{attribute 'linkalways'} 
{attribute 'no_explicit_call' := 'This FB is a CLASS and must be accessed using methods or properties'}
{attribute 'enable_dynamic_creation'}
FUNCTION_BLOCK _ALIASTYP EXTENDS AliasDatatypeBase
VAR
	localData : ALIASTYP;
	activeData : REFERENCE TO ALIASTYP REF= localData;
	aliasBaseDatatype : ALIASTYPBASE;
END_VAR

PROPERTY PUBLIC Address : PVOID
GET
Address := ADR(activeData);
END_GET
END_PROPERTY

METHOD PUBLIC ClearReference
VAR_INPUT
END_VAR
activeData REF= localData;
SetBaseDatatypeReference();
END_METHOD

METHOD PUBLIC Clone : I_Datatype
VAR
    pClone : POINTER TO _ALIASTYP;
END_VAR
pClone := __NEW(_ALIASTYP);
Clone := pClone^;
END_METHOD

METHOD FB_init : BOOL
VAR_INPUT
	bInitRetains : BOOL; // if TRUE, the retain variables are initialized (warm start / cold start)
	bInCopyCode : BOOL;  // if TRUE, the instance afterwards gets moved into the copy code (online change)
	//InitialValue : ALIASTYP; // if possible, not all values can be initialized
END_VAR
//localData := InitialValue; // if possible, not all values can be initialized
SetBaseDatatypeReference();
AddBaseDatatype(aliasBaseDatatype);
END_METHOD

PROPERTY PUBLIC Identifier : T_MAXSTRING
GET
Identifier := 'ALIASTYP';
END_GET
END_PROPERTY

METHOD PUBLIC MakeReferenceTo
VAR_INPUT
	ReferenceTarget : REFERENCE TO ALIASTYP;
END_VAR
activeData REF= ReferenceTarget;
SetBaseDatatypeReference();
END_METHOD

METHOD PROTECTED SetBaseDatatypeReference
VAR_INPUT
END_VAR
aliasBaseDatatype.MakeReferenceTo(activeData);
END_METHOD

PROPERTY PUBLIC Size : UDINT
GET
Size := SIZEOF(activeData);
END_GET
END_PROPERTY

METHOD TryMakeReferenceTo : BOOL
VAR_INPUT
	Target : I_Datatype;
END_VAR
VAR
	pTargetData : POINTER TO ALIASTYP;
END_VAR
IF NOT IsEquivalentTo(Target) THEN
	RETURN;
END_IF

pTargetData := Target.Address;
activeData REF= pTargetData^;
SetBaseDatatypeReference();
TryMakeReferenceTo := TRUE;
END_METHOD

PROPERTY PUBLIC Value : REFERENCE TO ALIASTYP
GET
Value REF= activeData;
END_GET
END_PROPERTY

END_FUNCTION_BLOCK

(* stored: Version 1.1.0.1, ProductVersion 3.1.4024.13
   POU _ALIASTYP: Id {11dfa79a-cf49-0cc9-1ff2-2a890e36ced1}, SpecialFunc None
   Folder Core: Id {cc189060-d94f-0946-012c-c0e35767e96e}
   Folder Protected: Id {62ce3d2f-1ab3-0f0b-1775-9976f8c1ba1c}
   Folder Customize: Id {1edd4a7a-953f-0d09-1983-04adff481ec5}
   Folder Constructor: Id {06f36322-8592-0889-1ecb-d2277949b744}
   Property Address: Id {acb4897b-300b-02f7-1574-3139e91f367e}
   Get Get: Id {cbb3e3b2-47c8-0f8e-2c9d-13790e1b607d}
   Method ClearReference: Id {5bbc1ba8-8dae-0042-2e39-57f033e9b97a}
   Method Clone: Id {382e9781-35fa-0f2d-1651-b5755299772d}
   Method FB_init: Id {3acb41ac-850d-05c9-1152-c4f120939b48}
   Property Identifier: Id {318825c9-d301-0c0d-32c8-5ec92b72736c}
   Get Get: Id {5e762c12-9b35-0e5c-299e-6cf69858a11e}
   Method MakeReferenceTo: Id {6259c631-a2d6-0426-1c5a-6fbc04d22a97}
   Method SetBaseDatatypeReference: Id {3f2077cb-c414-0424-0d19-16425e29d5f4}
   Property Size: Id {48dab08c-b54a-0b04-0498-02e2e93ee143}
   Get Get: Id {b23df07f-b43d-0936-2742-ac673b5494dc}
   Method TryMakeReferenceTo: Id {9b24dae1-36ca-00bf-0a54-29b6900c0a33}
   Property Value: Id {40375163-87b0-08ab-2945-36f111e497c6}
   Get Get: Id {4a4d920f-8f94-050f-1d7d-d1d77622d645} *)
